# B&R Automation Studio project Billy
Automation Studio 4.12.4.107 SP

## Configuration Config1

CPU PC_any, AutomationRuntime H4.93, Build 4.1.2, Vc V4.73.1

### Task classes (Cpu.sw)
```
Cyclic#1:
  TCPChatPrg <- BillyTests.TCPChatTest.prg
Binaries: FWRules, TCData, udbdef, asfw, User, iomap, sysconf, arconfig, ashwd, Role, ashwac
Libraries: AsTCP, runtime, Billy, asstring, asieccon, astime, MyTCPLib
```

### Hardware
```
PC : PC_any v1.1.1.0 (OrderNumber=PC)
  ConfigurationID = TCPIP_test_Config1
  FileDevice1
  FileDeviceName1 = USER
  FileDevicePath1 = USER_PATH
```

- Physical/Config1/PC/IoMap.iom: same as Physical/Config1/PC/Cpu.per
- Physical/Config1/PC/PvMap.vvm: same as Physical/Config1/PC/Cpu.per
- Safety project (password-protected, skipped)

## Logical view

Binary libraries used (declarations not repeated): operator, runtime, astime, AsIecCon, AsTCP, asstring

### Package Logical/Libraries - Global libraries

### Library Logical/Libraries/Billy (IEC) - This is Billy the most famous library library in the world!
Depends on: AsTCP, asstring

#### Billy.fun - Exported functions and function blocks
```iecst
FUNCTION_BLOCK TCPChatFB (*FB template for Enable FB*)
	VAR_INPUT
		Enable : BOOL; (*Enable the function block*)
		Update : BOOL; (*Update parameters*)
		Parameters : TCPChatParametersType; (*Parameter required for computing*)
		Reset : BOOL;
		MessageToSend : STRING[tcpchatMESSAGE_LEN]; (*Input variable*)
	END_VAR
	VAR_OUTPUT
		Active : BOOL; (*Function block is active*)
		Error : BOOL; (*Indicates an error*)
		StatusID : DINT; (*Status information*)
		MessageReceived : STRING[tcpchatMESSAGE_LEN]; (*Output variable*)
	END_VAR
	VAR
		Internal : TCPChatFBInternalType; (*Data for internal use*)
	END_VAR
END_FUNCTION_BLOCK
```

#### TCPChatFBConstants.var - Exported constants
```iecst
VAR CONSTANT
	tcpchatMESSAGE_LEN : UINT := 200;
	tcpchatMAX_CONNECTIONS_NUM : USINT := 32;
END_VAR
```

#### TCPChatFBTypes.typ - Exported data types
```iecst
TYPE
	TCPChatFBInternalType : 	STRUCT  (*Template of a structure of internal parameters for an enable function block *)
		Enabled : BOOL; (*Variable to detect rising edge on Enable input*)
		Updated : BOOL; (*Variable to detect rising edge of Update input*)
		Reseted : BOOL; (*Variable to detect rising edge of Reset input*)
		ParametersValid : BOOL; (*All parameters valid flag*)
		Parameters : TCPChatParametersType; (*Internal parameter for computing*)
		TcpOpenLocalInterface : TcpOpen; (*AsTCP.TcpOpen FUB*)
		TcpClientConnection : TcpClient; (*AsTCP.TcpClient FUB*)
		TcpReceiveMessage : TcpRecv; (*AsTCP.TcpRecv FUB*)
		TcpSendMessage : TcpSend; (*AsTCP.TcpSend FUB*)
		TcpCloseConnection : TcpClose; (*AsTCP.TcpClose FUB*)
		TcpServerInstance : TcpServer; (*AsTCP.TcpClose FUB*)
		MachineStateStep : UINT;
		SendingMessage : STRING[tcpchatMESSAGE_LEN];
		LastMessageSent : STRING[tcpchatMESSAGE_LEN];
		RetryOpenLocalCnt : USINT;
		RetryClientConnectionCnt : USINT;
		SocketIDs : ARRAY[0..tcpchatMAX_CONNECTIONS_NUM]OF UDINT;
	END_STRUCT;
	TCPChatParametersType : 	STRUCT
		ServerIPAddress : STRING[15];
		ServerPort : UINT;
		ServerRole : BOOL;
	END_STRUCT;
END_TYPE
```

#### TCPChatFB.st
```iecst
FUNCTION_BLOCK TCPChatFB

	IF Enable THEN

        IF NOT Internal.Enabled OR (Update AND NOT Internal.Updated) THEN
			TCPChatFBCheckParameters;
		END_IF;
		Internal.Updated := Update;

        IF Internal.ParametersValid THEN
            TCPChatFBCyclicCode;
        END_IF;

        Internal.Enabled := Enable;
    ELSE
        TCPChatFBResetInternal;
        TCPChatFBResetOutputs;
    END_IF;

END_FUNCTION_BLOCK
```

#### TCPChatFBActions.st
```iecst
ACTION TCPChatFBCheckParameters:
    IF strlen(ADR(Parameters.ServerIPAddress)) = 0 THEN
		StatusID := tcpERR_PARAMETER;
		Error := TRUE;
	ELSIF Parameters.ServerPort = 0 THEN
		StatusID := tcpERR_PARAMETER;
		Error := TRUE;
	ELSE
		Error := FALSE;
        Internal.Parameters := Parameters;
        Internal.ParametersValid := TRUE;
    END_IF;
END_ACTION

ACTION TCPChatFBCyclicClientCode:

	CASE Internal.MachineStateStep OF

		0: // Init
			StatusID := ERR_FUB_BUSY;

			TCPChatFBResetOutputs;

			Internal.RetryOpenLocalCnt := 0;
			Internal.RetryClientConnectionCnt := 0;

			memset(ADR(Internal.LastMessageSent),0,SIZEOF(Internal.LastMessageSent));

			Internal.MachineStateStep := 10;

		10: // Open Ethernet Interface
			StatusID := ERR_FUB_BUSY;

			Internal.TcpOpenLocalInterface.enable := TRUE;
			Internal.TcpOpenLocalInterface.pIfAddr := 0; // Client listen on all interfaces
			Internal.TcpOpenLocalInterface.port := 0; // A free port is asigned automatically
			Internal.TcpOpenLocalInterface.options := 0;
			Internal.TcpOpenLocalInterface();  // Call the Function

			IF Internal.TcpOpenLocalInterface.status = ERR_OK THEN
				Internal.SocketIDs[0] := Internal.TcpOpenLocalInterface.ident;
				Internal.RetryOpenLocalCnt := 0;
				Internal.MachineStateStep := 20;
			ELSIF Internal.TcpOpenLocalInterface.status = ERR_FUB_BUSY THEN
				// wait
			ELSIF Internal.TcpOpenLocalInterface.status = tcpERR_ALREADY_EXIST AND Internal.RetryOpenLocalCnt = 0 THEN
				Internal.SocketIDs[0] := Internal.TcpOpenLocalInterface.ident;
				Internal.RetryOpenLocalCnt := Internal.RetryOpenLocalCnt + 1;
				Internal.MachineStateStep := 11;
			ELSE
				StatusID := Internal.TcpOpenLocalInterface.status;
				Internal.MachineStateStep := 99;
			END_IF

		11: // Close socket due to an error -> after this state it retries to establish a connection
			StatusID := ERR_FUB_BUSY;

			Internal.TcpCloseConnection.enable := TRUE;
			Internal.TcpCloseConnection.ident := Internal.SocketIDs[0];
			Internal.TcpCloseConnection.how := 0;
			Internal.TcpCloseConnection();

			IF Internal.TcpCloseConnection.status <> ERR_FUB_BUSY THEN
				Internal.SocketIDs[0] := 0;
				Internal.MachineStateStep := 10;
			END_IF

		20: // Connect to the other Station
			StatusID := ERR_FUB_BUSY;

			Internal.TcpClientConnection.enable := TRUE;
			Internal.TcpClientConnection.ident := Internal.SocketIDs[0];
			Internal.TcpClientConnection.portserv := Internal.Parameters.ServerPort;
			Internal.TcpClientConnection.pServer := ADR(Internal.Parameters.ServerIPAddress);
			Internal.TcpClientConnection();

			IF Internal.TcpClientConnection.status = ERR_OK THEN
				Internal.RetryClientConnectionCnt := 0;
				Internal.MachineStateStep := 30;
			ELSIF Internal.TcpClientConnection.status = ERR_FUB_BUSY THEN
				// wait
			ELSIF Internal.TcpClientConnection.status = tcpERR_ALREADY_CONNECTED AND Internal.RetryClientConnectionCnt = 0 THEN
				Internal.RetryClientConnectionCnt := Internal.RetryClientConnectionCnt + 1;
				Internal.MachineStateStep := 11;
			ELSIF Internal.TcpClientConnection.status = tcpERR_INVALID THEN  // wait server
				// wait
			ELSE
				StatusID := Internal.TcpClientConnection.status;
				Internal.MachineStateStep := 99;
			END_IF

		30: // Wait a message to be sent and listen for message from server
			StatusID := ERR_OK;

			IF MessageToSend <> Internal.LastMessageSent THEN // Check if a new message is waiting to be sent
				IF strlen(ADR(MessageToSend)) > 0 THEN
					Internal.SendingMessage := MessageToSend;
					Internal.MachineStateStep := 40;
				ELSE
					Internal.LastMessageSent := MessageToSend;
				END_IF

			ELSE
				Internal.TcpReceiveMessage.enable := TRUE;
				Internal.TcpReceiveMessage.ident := Internal.SocketIDs[0];
				Internal.TcpReceiveMessage.pData := ADR(MessageReceived);
				Internal.TcpReceiveMessage.datamax := SIZEOF(MessageReceived);
				Internal.TcpReceiveMessage.flags := 0;
				Internal.TcpReceiveMessage();

				IF Internal.TcpReceiveMessage.status = ERR_OK THEN
					// do nothing
				ELSIF Internal.TcpReceiveMessage.status = tcpERR_NO_DATA THEN
					// do nothing
				ELSIF Internal.TcpReceiveMessage.status = ERR_FUB_BUSY THEN
					// wait
				ELSIF Internal.TcpReceiveMessage.status = tcpERR_NOT_CONNECTED THEN
					Internal.MachineStateStep := 11;
				ELSE
					StatusID := Internal.TcpReceiveMessage.status;
					Internal.MachineStateStep := 99;
				END_IF
			END_IF

		40: // Send Data to the Server
			StatusID := ERR_FUB_BUSY;

			Internal.TcpSendMessage.enable := TRUE;
			Internal.TcpSendMessage.ident := Internal.SocketIDs[0];
			Internal.TcpSendMessage.pData := ADR(Internal.SendingMessage);
			Internal.TcpSendMessage.datalen := SIZEOF(Internal.SendingMessage);
			Internal.TcpSendMessage.flags := 0;
			Internal.TcpSendMessage();

			IF Internal.TcpSendMessage.status = ERR_OK THEN
				Internal.LastMessageSent := Internal.SendingMessage;
				Internal.MachineStateStep := 30;
			ELSIF Internal.TcpSendMessage.status = ERR_FUB_BUSY THEN
				// wait
			ELSIF Internal.TcpSendMessage.status = tcpERR_NOT_CONNECTED THEN
				Internal.MachineStateStep := 11;
			ELSE
				StatusID := Internal.TcpSendMessage.status;
				Internal.MachineStateStep := 99;
			END_IF

		99: // An error occured -> close connection and go to error state
			IF Internal.SocketIDs[0] <> 0 THEN
				Internal.TcpCloseConnection.enable := TRUE;
				Internal.TcpCloseConnection.ident := Internal.SocketIDs[0];
				Internal.TcpCloseConnection.how := 0;
				Internal.TcpCloseConnection();

				IF Internal.TcpCloseConnection.status <> ERR_FUB_BUSY THEN
					Internal.SocketIDs[0] := 0;
				END_IF
			ELSE

				IF Reset AND NOT Internal.Reseted THEN
					Internal.Reseted := TRUE;
					Internal.MachineStateStep := 0;
				END_IF
			END_IF

		ELSE
			Internal.MachineStateStep := 0;

	END_CASE

	IF NOT Reset THEN
		Internal.Reseted := FALSE;
	END_IF

	Active := Internal.MachineStateStep = 30 OR Internal.MachineStateStep = 40;
	Error := Internal.MachineStateStep = 99;
END_ACTION

ACTION TCPChatFBCyclicServerCode:
	CASE Internal.MachineStateStep OF

		0: // Init
			StatusID := ERR_FUB_BUSY;

			TCPChatFBResetOutputs;

			Internal.RetryOpenLocalCnt := 0;
			Internal.RetryClientConnectionCnt := 0;

			memset(ADR(Internal.LastMessageSent),0,SIZEOF(Internal.LastMessageSent));
			memset(ADR(Internal.SocketIDs),0,SIZEOF(Internal.SocketIDs));

			Internal.MachineStateStep := 10;

		10: // Open Ethernet Interface
			StatusID := ERR_FUB_BUSY;

			Internal.TcpOpenLocalInterface.enable := TRUE;
			Internal.TcpOpenLocalInterface.pIfAddr := 0; // Client listen on all interfaces
			Internal.TcpOpenLocalInterface.port := 0; // A free port is asigned automatically
			Internal.TcpOpenLocalInterface.options := 0;
			Internal.TcpOpenLocalInterface();  // Call the Function

			IF Internal.TcpOpenLocalInterface.status = ERR_OK THEN
				Internal.SocketIDs[0] := Internal.TcpOpenLocalInterface.ident;
				Internal.RetryOpenLocalCnt := 0;
				Internal.MachineStateStep := 20;
			ELSIF Internal.TcpOpenLocalInterface.status = ERR_FUB_BUSY THEN
				// wait
			ELSIF Internal.TcpOpenLocalInterface.status = tcpERR_ALREADY_EXIST AND Internal.RetryOpenLocalCnt = 0 THEN
				Internal.SocketID := Internal.TcpOpenLocalInterface.ident;
				Internal.RetryOpenLocalCnt := Internal.RetryOpenLocalCnt + 1;
				Internal.MachineStateStep := 11;
			ELSE
				StatusID := Internal.TcpOpenLocalInterface.status;
				Internal.MachineStateStep := 99;
			END_IF

		11: // Close socket due to an error -> after this state it retries to establish a connection
			StatusID := ERR_FUB_BUSY;

			Internal.TcpCloseConnection.enable := TRUE;
			Internal.TcpCloseConnection.ident := Internal.SocketIDs[0];
			Internal.TcpCloseConnection.how := 0;
			Internal.TcpCloseConnection();

			IF Internal.TcpCloseConnection.status <> ERR_FUB_BUSY THEN
				Internal.SocketIDs[0] := 0;
				Internal.MachineStateStep := 10;
			END_IF

		20: // Connect to the other Station
			StatusID := ERR_FUB_BUSY;

			Internal.TcpServerInstance.enable := TRUE;
			Internal.TcpServerInstance.ident := Internal.SocketIDs[0];
			Internal.TcpServerInstance.backlog := 1;
			Internal.TcpServerInstance.portserv := Internal.Parameters.ServerPort;
			Internal.TcpServerInstance.pServer := ADR(Internal.Parameters.ServerIPAddress);
			Internal.TcpServerInstance();

			IF Internal.TcpClientConnection.status = ERR_OK THEN
				Internal.RetryClientConnectionCnt := 0;
				Internal.MachineStateStep := 30;
			ELSIF Internal.TcpClientConnection.status = ERR_FUB_BUSY THEN
				// wait
			ELSIF Internal.TcpClientConnection.status = tcpERR_ALREADY_CONNECTED AND Internal.RetryClientConnectionCnt = 0 THEN
				Internal.RetryClientConnectionCnt := Internal.RetryClientConnectionCnt + 1;
				Internal.MachineStateStep := 11;
			ELSIF Internal.TcpClientConnection.status = tcpERR_INVALID THEN  // wait server
				// wait
			ELSE
				StatusID := Internal.TcpClientConnection.status;
				Internal.MachineStateStep := 99;
			END_IF

		30: // Wait a message to be sent and listen for message from server
			StatusID := ERR_OK;

			IF MessageToSend <> Internal.LastMessageSent THEN // Check if a new message is waiting to be sent
				IF strlen(ADR(MessageToSend)) > 0 THEN
					Internal.SendingMessage := MessageToSend;
					Internal.MachineStateStep := 40;
				ELSE
					Internal.LastMessageSent := MessageToSend;
				END_IF

			ELSE
				Internal.TcpReceiveMessage.enable := TRUE;
				Internal.TcpReceiveMessage.ident := Internal.SocketID;
				Internal.TcpReceiveMessage.pData := ADR(MessageReceived);
				Internal.TcpReceiveMessage.datamax := SIZEOF(MessageReceived);
				Internal.TcpReceiveMessage.flags := 0;
				Internal.TcpReceiveMessage();

				IF Internal.TcpReceiveMessage.status = ERR_OK THEN
					// do nothing
				ELSIF Internal.TcpReceiveMessage.status = tcpERR_NO_DATA THEN
					// do nothing
				ELSIF Internal.TcpReceiveMessage.status = ERR_FUB_BUSY THEN
					// wait
				ELSIF Internal.TcpReceiveMessage.status = tcpERR_NOT_CONNECTED THEN
					Internal.MachineStateStep := 11;
				ELSE
					StatusID := Internal.TcpReceiveMessage.status;
					Internal.MachineStateStep := 99;
				END_IF
			END_IF

		40: // Send Data to the Server
			StatusID := ERR_FUB_BUSY;

			Internal.TcpSendMessage.enable := TRUE;
			Internal.TcpSendMessage.ident := Internal.SocketID;
			Internal.TcpSendMessage.pData := ADR(Internal.SendingMessage);
			Internal.TcpSendMessage.datalen := SIZEOF(Internal.SendingMessage);
			Internal.TcpSendMessage.flags := 0;
			Internal.TcpSendMessage();

			IF Internal.TcpSendMessage.status = ERR_OK THEN
				Internal.LastMessageSent := Internal.SendingMessage;
				Internal.MachineStateStep := 30;
			ELSIF Internal.TcpSendMessage.status = ERR_FUB_BUSY THEN
				// wait
			ELSIF Internal.TcpSendMessage.status = tcpERR_NOT_CONNECTED THEN
				Internal.MachineStateStep := 11;
			ELSE
				StatusID := Internal.TcpSendMessage.status;
				Internal.MachineStateStep := 99;
			END_IF

		99: // An error occured -> close connection and go to error state
			IF Internal.SocketID <> 0 THEN
				Internal.TcpCloseConnection.enable := TRUE;
				Internal.TcpCloseConnection.ident := Internal.SocketID;
				Internal.TcpCloseConnection.how := 0;
				Internal.TcpCloseConnection();

				IF Internal.TcpCloseConnection.status <> ERR_FUB_BUSY THEN
					Internal.SocketID := 0;
				END_IF
			ELSE

				IF Reset AND NOT Internal.Reseted THEN
					Internal.Reseted := TRUE;
					Internal.MachineStateStep := 0;
				END_IF
			END_IF

		ELSE
			Internal.MachineStateStep := 0;

	END_CASE

	IF NOT Reset THEN
		Internal.Reseted := FALSE;
	END_IF

	Active := Internal.MachineStateStep = 30 OR Internal.MachineStateStep = 40;
	Error := Internal.MachineStateStep = 99;
END_ACTION

ACTION TCPChatFBCyclicCode:

	IF Internal.Parameters.ServerRole THEN
		TCPChatFBCyclicServerCode;
	ELSE
		TCPChatFBCyclicClientCode;
	END_IF

END_ACTION

ACTION TCPChatFBResetInternal:

	IF Internal.SocketID <> 0 THEN // An open connection exists -> close it
		Internal.TcpCloseConnection.enable := TRUE;
		Internal.TcpCloseConnection.ident := Internal.SocketID;
		Internal.TcpCloseConnection.how := 0;
		Internal.TcpCloseConnection();

		IF Internal.TcpCloseConnection.status <> ERR_FUB_BUSY THEN
			Internal.SocketID := 0;
		END_IF
	ELSE

		memset(ADR(Internal.Parameters),0,SIZEOF(Internal.Parameters));
		memset(ADR(Internal.SocketIDs),0,SIZEOF(Internal.SocketIDs));
		Internal.Enabled := FALSE;
		Internal.ParametersValid := FALSE;
		Internal.MachineStateStep := 0;

	END_IF

END_ACTION

ACTION TCPChatFBResetOutputs:

	Active := FALSE;
	Error := FALSE;
	StatusID := 0;
	MessageReceived := '';

END_ACTION
```

### Program Logical/BillyTests/TCPChatTest (IEC)

#### Main.st - Init, cyclic, exit code
```iecst
PROGRAM _INIT
	TcpChat1.Parameters.ServerIPAddress := '127.0.0.1';
	TcpChat1.Parameters.ServerPort := 12000;
	TcpChat1.Parameters.ServerRole := FALSE;

	TcpChat2.Parameters.ServerIPAddress := '127.0.0.1';
	TcpChat2.Parameters.ServerPort := 12000;
	TcpChat2.Parameters.ServerRole := TRUE;
END_PROGRAM

PROGRAM _CYCLIC
	TcpChat1();
	TcpChat2();
END_PROGRAM

PROGRAM _EXIT

END_PROGRAM
```

#### Variables.var - Local variables
```iecst
VAR
	TcpChat1 : TCPChatFB;
	TcpChat2 : TCPChatFB;
END_VAR
```
